// TIA Portal V20 export
DATA_BLOCK "CM_Name"   // DB105
// stored: Access Published, MemoryReserve 100, Namespace Unit1
   VAR
      ReadFromHMI : Bool;
      WriteToHMI : Bool;
      AxisName : Array[1..45] of WString [25];
      CylinderName : Array[1..50] of WString [25];
      VaccName : Array[1..25] of WString [25];
   END_VAR
BEGIN
   AxisName[1] := WSTRING#'';   // UnwinderTopAxisB
   AxisName[2] := WSTRING#'';   // UnwinderBottomAxisB
   AxisName[3] := WSTRING#'';   // compenastor X
   AxisName[4] := WSTRING#'';
   AxisName[5] := WSTRING#'';   // AnodeMainPnP1AxisX
   AxisName[6] := WSTRING#'';   // AnodeMainPnP2AxisX
   AxisName[7] := WSTRING#'';   // CathodeMainPnP1AxisX
   AxisName[8] := WSTRING#'';   // CathodeMainPnP2AxisX
   AxisName[9] := WSTRING#'';   // CathodeMainPnP1AxisY
   AxisName[10] := WSTRING#'';   // CathodeMainPnP1AxisZ
   AxisName[11] := WSTRING#'';   // AnodeMainPnP1AxisY
   AxisName[12] := WSTRING#'';   // AnodeMainPnP1AxisZ
   AxisName[13] := WSTRING#'';   // CathodeMainPnP2AxisZ
   AxisName[14] := WSTRING#'';   // AnodeMainPnP2AxisZ
   AxisName[15] := WSTRING#'';   // AnodeAlignTableAxisX
   AxisName[16] := WSTRING#'';   // AnodeAlignTableAxisY1
   AxisName[17] := WSTRING#'';   // AnodeAlignTableAxisY2
   AxisName[18] := WSTRING#'';   // CathodeAlignTableAxisX
   AxisName[19] := WSTRING#'';   // CathodeAlignTableAxisY1
   AxisName[20] := WSTRING#'';   // CathodeAlignTableAxisY2
   AxisName[21] := WSTRING#'';   // FinalRollerFrontAxisX
   AxisName[22] := WSTRING#'';   // FinalRollerRearAxisX
   AxisName[23] := WSTRING#'';   // MandrelFLAxisY
   AxisName[24] := WSTRING#'';   // MandrelFLAxisZ
   AxisName[25] := WSTRING#'';   // MandrelFRAxisY
   AxisName[26] := WSTRING#'';   // MandrelFRAxisZ
   AxisName[27] := WSTRING#'';   // MandrelRLAxisY
   AxisName[28] := WSTRING#'';   // MandrelRLAxisZ
   AxisName[29] := WSTRING#'';   // MandrelRRAxisY
   AxisName[30] := WSTRING#'';   // MandrelRRAxisZ
   AxisName[31] := WSTRING#'';   // StackTableAxisZ
   AxisName[32] := WSTRING#'';   // StackTableOutFrontAxisZ
   AxisName[33] := WSTRING#'';   // StackTableOutRearAxisZ
   AxisName[34] := WSTRING#'';   // SepaClampnCutterAxisX
   AxisName[35] := WSTRING#'';   // SepaClampnCutterAxisZ
   AxisName[36] := WSTRING#'';   // SepaGripperAxisX
   AxisName[37] := WSTRING#'';   // SepaGripperAxisZ
   AxisName[38] := WSTRING#'';   // SepaGripperAxisC
   AxisName[39] := WSTRING#'';   // JRWinderFrontAxisY
   AxisName[40] := WSTRING#'';   // JRWinderRearAxisY
   AxisName[41] := WSTRING#'';   // JRWinderAxisB
   CylinderName[1] := WSTRING#'';   // UnwinderAirShaftTop
   CylinderName[2] := WSTRING#'';   // UnwinderAirShaftBottom
   CylinderName[3] := WSTRING#'';   // SuctionPadTopUpDown
   CylinderName[4] := WSTRING#'';   // SuctionPadBtmUpDown
   CylinderName[5] := WSTRING#'';   // CutterUpDown
   CylinderName[6] := WSTRING#'';   // TapeTopUpDown
   CylinderName[7] := WSTRING#'';   // TapeBtmUpDown
   CylinderName[8] := WSTRING#'';   // SpliceHeadRotateTopFwdBwd
   CylinderName[9] := WSTRING#'';   // SpliceHeadRotateBtmFwdBwd
   CylinderName[10] := WSTRING#'';   // DancerFwdBwd
   CylinderName[11] := WSTRING#'';   // SepaUnwinderIonizer
   CylinderName[12] := WSTRING#'';   // SepaUnwinderIonizerBottom
   CylinderName[13] := WSTRING#'';   // AnodeNgBoxLiftUpDown
   CylinderName[14] := WSTRING#'';
   CylinderName[15] := WSTRING#'';   // AnodeNgBoxLockUpDown
   CylinderName[16] := WSTRING#'';   // AnodeMaintenanceMovingFixFrontFwdBwd
   CylinderName[17] := WSTRING#'';   // AnodeGlassCleaning
   CylinderName[18] := WSTRING#'';   // AnodeNgPnp1stFwdBwd
   CylinderName[19] := WSTRING#'';   // AnodeNgPnpUpDown
   CylinderName[20] := WSTRING#'';
   CylinderName[21] := WSTRING#'';   // AnodeMainPnP1RotaryCwCcw
   CylinderName[22] := WSTRING#'';   // AnodeNgPnp2ndFwdBwd
   CylinderName[23] := WSTRING#'';   // CathodeMaintenanceMovingFixFrontFwdBwd
   CylinderName[24] := WSTRING#'';
   CylinderName[25] := WSTRING#'';   // CathodeNgBoxLockUpDown
   CylinderName[26] := WSTRING#'';   // CathodeNgBoxLiftUpDown
   CylinderName[27] := WSTRING#'';   // CathodeNgPnp2ndFwdBwd
   CylinderName[28] := WSTRING#'';
   CylinderName[29] := WSTRING#'';   // CathodeNgPnpUpDown
   CylinderName[30] := WSTRING#'';   // CathodeGlassCleaning
   CylinderName[31] := WSTRING#'';   // CathodeMainPnP1RotaryCwCcw
   CylinderName[32] := WSTRING#'';   // CathodeNgPnp1stFwdBwd
   CylinderName[33] := WSTRING#'';   // MendrelFLClamp
   CylinderName[34] := WSTRING#'';   // MendrelFRClamp
   CylinderName[35] := WSTRING#'';   // MendrelRLClamp
   CylinderName[36] := WSTRING#'';   // MendrelRRClamp
   CylinderName[37] := WSTRING#'';   // StackTableGapPadUpDown
   CylinderName[38..39] := WSTRING#'';
   CylinderName[40] := WSTRING#'';   // JRWinderClampRightBtmUpDown
   CylinderName[41] := WSTRING#'';   // JRWinderClampLeftBtmUpDown
   CylinderName[42] := WSTRING#'';   // JRWinderClampLeftTopUpDown
   CylinderName[43] := WSTRING#'';   // StackGripperFwdBwd
   CylinderName[44] := WSTRING#'';   // SepaClampBottomUpDown
   CylinderName[45] := WSTRING#'';   // SepaClampTopUpDown
   CylinderName[46] := WSTRING#'';   // SepaCutterLeftUpDown
   CylinderName[47] := WSTRING#'';   // JRWinderClampRightTopUpDown
   CylinderName[48..49] := WSTRING#'';
   VaccName[1] := WSTRING#'';   // cmSuctionPadTopLeftVaccum
   VaccName[2] := WSTRING#'';   // cmSuctionPadTopRightVaccum
   VaccName[3] := WSTRING#'';   // cmSuctionPadBtmLeftVaccum
   VaccName[4] := WSTRING#'';   // cmSuctionPadBtmRightVaccum
   VaccName[5] := WSTRING#'';   // cmSuctionPadTopTapeVaccum
   VaccName[6] := WSTRING#'';   // cmSuctionPadBtmTapeVaccum
   VaccName[7..9] := WSTRING#'';
   VaccName[10] := WSTRING#'';   // cmAnodeMainPnP1SuctionPlateVacuum
   VaccName[11] := WSTRING#'';   // cmAnodeMainPnP2SuctionPlateVacuum
   VaccName[12] := WSTRING#'';   // cmAnodeAlignTableSuctionPlateVacuum
   VaccName[13] := WSTRING#'';   // cmAnodeNgPnpVaccum
   VaccName[14] := WSTRING#'';
   VaccName[15] := WSTRING#'';   // cmCathodeMainPnP1SuctionPlateVacuum
   VaccName[16] := WSTRING#'';   // cmCathodeMainPnP2SuctionPlateVacuum
   VaccName[17] := WSTRING#'';   // cmCathodeAlignTableSuctionPlateVacuum
   VaccName[18] := WSTRING#'';   // cmCathodeNgPnpVaccum
   VaccName[19] := WSTRING#'';
   VaccName[20] := WSTRING#'';   // cmStackTableVaccum
   VaccName[21..25] := WSTRING#'';
END_DATA_BLOCK
